// TIA Portal V20 export
TYPE "typeEm1Standard"
// stored: Access Published, Namespace Unit1
   STRUCT
      commands { ExternalWritable := 'False'} : "Unit1.typeEm1Commands";
      monitoring { ExternalWritable := 'False'} : "Unit1.typeEm1Monitoring";
   END_STRUCT;
END_TYPE
